INTERFACE ITF_HMIConfiguration

METHOD MainMenuConfigure : BOOL
VAR_INPUT
	itfHMIManager			: ITF_HMIManagerConfigure;
END_VAR
END_METHOD

END_INTERFACE

(* stored: Version 1.1.0.1
   Itf ITF_HMIConfiguration: Id {d7340403-e938-4a39-b0ea-a459eb342446}
   Method MainMenuConfigure: Id {1e0869f0-3d07-0b3c-0db2-39d4e328e682} *)
